// A function block for TcpIp control. Body should be called, 
// but all the logic is done with method calling and awaiting "TRUE" returned when the method finishes.
FUNCTION_BLOCK FB_TcpIpCommControl 
EXTENDS ZigaLibs_Core.FB_HasInstanceNameAndPath 
IMPLEMENTS I_TcpIpCommControl

VAR
	_socketClose			: Tc2_TcpIp.FB_SocketClose;
	_error					: BOOL;
	_errorReceiving			: BOOL;
	_errorSending			: BOOL;
	_isConnected			: BOOL;
	_clientServerControl	: Tc2_TcpIp.FB_ClientServerConnection;
	_socketHandle			: Tc2_TcpIp.T_HSOCKET;
	_logger					: REFERENCE TO ZigaLibs_Logging.I_Logger;
END_VAR

_clientServerControl(nMode := Tc2_TcpIp.CONNECT_MODE_ENABLEDBG, hSocket => _socketHandle);
_error := _errorReceiving OR _errorSending OR _clientServerControl.bError;

// Connets to the target client with the provided Ip address and port
METHOD Connect : BOOL
VAR_INPUT
	Ipv4Address	: Tc2_System.T_IPv4Addr;	// Ip Address
	Port		: UINT;	// Port
END_VAR
VAR_INST
	connected	: R_TRIG;
END_VAR
VAR
	sb	: ZigaLibs_Core.FB_StringBuilder;
END_VAR
connected(CLK := _clientServerControl.eState = Tc2_TcpIp.E_SocketConnectionState.eSOCKET_CONNECTED AND NOT _clientServerControl.bError);
IF connected.Q THEN
	sb.AddString('Connected to')
		.AddWithQuotationMark(_clientServerControl.sRemoteHost)
		.AddString(' with port ')
		.AddAny(_clientServerControl.nRemotePort);
	THIS^.WriteInfoLog(sb.Create());
END_IF

IF THIS^.IsConnected = FALSE THEN
	_clientServerControl.bEnable := TRUE;
	_clientServerControl.sRemoteHost := Ipv4Address;
	_clientServerControl.nRemotePort := Port;
	_clientServerControl.sSrvNetID := '';
ELSE
	Connect := TRUE;
END_IF
END_METHOD

// Disconnects from the server and closes all active socket connections. Returns TRUE when done.
METHOD Disconnect : BOOL
VAR_INST
	disconnected	: Tc2_Standard.F_TRIG;
END_VAR
VAR
	sb			: ZigaLibs_Core.FB_StringBuilder;
END_VAR
disconnected(CLK := _socketClose.bBusy AND NOT _socketClose.bError);
IF disconnected.Q THEN
	sb.AddString('Disconnected from ')
		.AddWithQuotationMark(_clientServerControl.sRemoteHost)
		.AddString(' with port ')
		.AddAny(_clientServerControl.nRemotePort);
	THIS^.WriteInfoLog(sb.Create());
END_IF

IF _clientServerControl.bEnable THEN
	_clientServerControl.bEnable := FALSE;
END_IF

IF NOT _socketClose.bBusy AND (_socketHandle.handle <> 0) THEN
	_socketClose(bExecute := TRUE, sSrvNetId := '', hSocket := _socketHandle);
END_IF
_socketClose(bExecute := FALSE, sSrvNetId := '', hSocket := _socketHandle);
_errorSending := FALSE;
_errorReceiving := FALSE;

Disconnect := NOT _socketClose.bBusy;
END_METHOD

{attribute 'monitoring' := 'call'}
PROPERTY Error : BOOL
GET
Error := _error;
END_GET
END_PROPERTY

METHOD FB_init : BOOL
VAR_INPUT
	bInitRetains 	: BOOL; // if TRUE, the retain variables are initialized (warm start / cold start)
	bInCopyCode 	: BOOL;  // if TRUE, the instance afterwards gets moved into the copy code (online change)
	logger			: REFERENCE TO ZigaLibs_Logging.I_Logger;
END_VAR
_logger REF= logger;
END_METHOD

METHOD GetLogPrefix : STRING
VAR_INPUT
END_VAR
GetLogPrefix := Tc2_Standard.CONCAT(THIS^.InstancePath, ': ');
END_METHOD

{attribute 'monitoring' := 'call'}
PROPERTY PUBLIC IsConnected : BOOL
GET
IsConnected := _clientServerControl.eState = Tc2_TcpIp.E_SocketConnectionState.eSOCKET_CONNECTED;
END_GET
END_PROPERTY

// Awaits a response from the client and returns TRUE when done. Response string can be found in the refResponse
// Method needs to be called untill TRUE is returned to finish the sending sequence!
METHOD Receive : BOOL
VAR_INPUT
	refResponse	: REFERENCE TO Tc2_System.T_MaxString;	// Response will be written to the string variable here
END_VAR
VAR_INST
	sResponse			: Tc2_System.T_MaxString;
	eSocketReceiveState	: E_SocketReceiveState;
	fbSocketReceive		: Tc2_TcpIp.FB_SocketReceive;
	bReceiveError		: BOOL;
END_VAR
VAR
	sb	: ZigaLibs_Core.FB_StringBuilder;
END_VAR
CASE eSocketReceiveState OF
	E_SocketReceiveState.READY:
		fbSocketReceive(bExecute := FALSE);
		IF THIS^.IsConnected THEN
			bReceiveError := FALSE;
			fbSocketReceive(
				bExecute := TRUE,
				cbLen := SIZEOF(refResponse),
				pDest := ADR(refResponse),
				sSrvNetId := '',
				hSocket := _socketHandle);
			eSocketReceiveState := E_SocketReceiveState.RECEIVING;
		END_IF
	
	E_SocketReceiveState.RECEIVING:
		fbSocketReceive(bExecute := FALSE);
		IF NOT fbSocketReceive.bError AND_THEN NOT fbSocketReceive.bBusy THEN
			eSocketReceiveState := E_SocketReceiveState.DONE;
		ELSIF fbSocketReceive.bError THEN
			eSocketReceiveState := E_SocketReceiveState.ERROR;	
		END_IF
	
	E_SocketReceiveState.DONE:
		Receive := TRUE;
		eSocketReceiveState := E_SocketReceiveState.READY;
	
	E_SocketReceiveState.ERROR:
		bReceiveError := TRUE;
		eSocketReceiveState := E_SocketReceiveState.DONE;
		
		sb.AddString('Error while receiving from ')
			.AddWithDblQuotationMarks(_socketHandle.remoteAddr.sAddr)
			.AddString('. Error code received is ')
			.AddWithQuotationMark(TO_STRING(fbSocketReceive.nErrId));
		THIS^.WriteErrorLog(sb.Create());
END_CASE

_errorReceiving := bReceiveError;
END_METHOD

{attribute 'monitoring' := 'call'}
(* Gets or sets the reconnect period. 
The value should not be set too low, since timeout periods of > 30 s may occur in the event of a network interruption. 
If the value is too low, command execution would be interrupted prematurely, and ADS error code 1861 (timeout elapsed) 
would be returned instead of the Winsocket error WSAETIMEDOUT.*)
PROPERTY PUBLIC ReconnectPeriod : TIME
GET
ReconnectPeriod := _clientServerControl.tReconnect;
END_GET
SET
IF ReconnectPeriod > T#30S THEN
	_clientServerControl.tReconnect := ReconnectPeriod;
END_IF
END_SET
END_PROPERTY

// Sends the command to the client and returns TRUE when done. 
// Method needs to be called untill TRUE is returned to finish the sending sequence!
METHOD Send : BOOL
VAR_INPUT
	sCommand	: Tc2_System.T_MaxString;	// Command to be send
END_VAR
VAR_INST
	fbSocketSend		: Tc2_TcpIp.FB_SocketSend;
	eSsocketSendState	: E_SocketSendState;
	arrSendDataBytes	: ARRAY[0..255] OF BYTE;
	nSendDataCount		: UDINT;
	bSendError			: BOOL;
END_VAR

VAR
	sb	: ZigaLibs_Core.FB_StringBuilder;
END_VAR
CASE eSsocketSendState OF
	E_SocketSendState.READY:
		bSendError := FALSE;
		IF sCommand <> '' THEN
			// Clear array for new data
			Tc2_System.MEMSET(
				destAddr := ADR(arrSendDataBytes),
				n := SIZEOF(arrSendDataBytes),
				fillByte := 0);
				
			// Prepare data
			Tc2_System.MEMCPY(
				destAddr := ADR(arrSendDataBytes),
				n := SIZEOF(sCommand),
				srcAddr := ADR(sCommand));
				
			// Get the data count, no empty bytes
			nSendDataCount := 0;
			FOR nSendDataCount := 0 TO SIZEOF(arrSendDataBytes) BY 1 DO
				IF arrSendDataBytes[nSendDataCount] = 0 THEN
					EXIT;
				END_IF
			END_FOR

			// Send data
			fbSocketSend(
				bExecute := TRUE,
				cbLen := nSendDataCount,
				pSrc := ADR(arrSendDataBytes),
				hSocket := _socketHandle);
				
			eSsocketSendState := E_SocketSendState.SENDING;
		END_IF
	
	E_SocketSendState.SENDING:
		fbSocketSend(bExecute := FALSE);
		IF fbSocketSend.bError THEN 
			eSsocketSendState := E_SocketSendState.ERROR;
		ELSIF fbSocketSend.bBusy = FALSE THEN
				eSsocketSendState := E_SocketSendState.DONE;
		END_IF
		
	E_SocketSendState.DONE:
		Send := TRUE;
		eSsocketSendState := E_SocketSendState.READY;
		
	E_SocketSendState.ERROR:
		bSendError := TRUE;
		eSsocketSendState := E_SocketSendState.DONE;
		sb.AddString('Error while sending from ')
			.AddWithQuotationMark(_socketHandle.localAddr.sAddr)
			.AddString(' to ')
			.AddWithDblQuotationMarks(_socketHandle.remoteAddr.sAddr)
			.AddString('. Command being sent was ')
			.AddWithQuotationMark(sCommand)
			.AddString('. Error code received is ')
			.AddWithQuotationMark(TO_STRING(fbSocketSend.nErrId));
		THIS^.WriteErrorLog(sb.Create());
		
END_CASE

_errorSending := bSendError;
END_METHOD

METHOD WriteErrorLog
VAR_INPUT
	message	: Tc2_System.T_MaxString;
END_VAR
IF NOT __ISVALIDREF(_logger) THEN
	RETURN;
END_IF

_logger.LogError(Tc2_Standard.CONCAT(THIS^.GetLogPrefix(), (message)));
END_METHOD

METHOD WriteInfoLog
VAR_INPUT
	message	: Tc2_System.T_MaxString;
END_VAR
IF NOT __ISVALIDREF(_logger) THEN
	RETURN;
END_IF

_logger.LogInfo(Tc2_Standard.CONCAT(THIS^.GetLogPrefix(), (message)));
END_METHOD

END_FUNCTION_BLOCK

(* stored: Version 1.1.0.1, ProductVersion 3.1.4024.15
   POU FB_TcpIpCommControl: Id {c1a18772-55c5-40c9-9a81-d2bef65ca48e}, SpecialFunc None
   Folder Constructor: Id {8e03ba55-7e0e-08dc-121d-63148ed4730e}
   Folder Private: Id {2efa374f-f01f-026b-1d46-811c1330f5ed}
   Folder Methods: Id {e8932037-c29c-0039-0710-e32b2dab25e8}
   Folder Public: Id {fad2bedc-c621-0e7a-10b3-e31e1f06606d}
   Folder Methods: Id {ca322448-3c94-05d4-3845-31017722f3e8}
   Folder Properties: Id {22abed52-9456-006d-1b18-e9ce2512ef08}
   Method Connect: Id {dd6866c4-171a-4bfc-95da-36f23ef555cb}
   Method Disconnect: Id {ed43bf91-0d1a-4937-b486-9810fb451075}
   Property Error: Id {5c00ee02-56f4-43bb-9e23-9bd70a569756}
   Get Get: Id {6ff5fc3c-9cf5-40c2-8121-3ea148df9e2e}
   Method FB_init: Id {7ffdea42-4472-0096-2bdd-6e582451a91a}
   Method GetLogPrefix: Id {18ab9aea-3da0-09f1-3eba-322fd828d465}
   Property IsConnected: Id {5e9ad8a1-6ad5-4c8b-a48a-e8e88fb474a1}
   Get Get: Id {d7cb8efd-ba1c-4704-9fa9-84315798b314}
   Method Receive: Id {7a2e245a-21db-4c97-a338-d1db7e183060}
   Property ReconnectPeriod: Id {960f0c0e-a8f0-4b6e-8253-4e69f0060513}
   Get Get: Id {873b00e4-9119-45cc-8128-e1136d45c726}
   Set Set: Id {6a4a98a9-2fc1-42f2-81eb-5c784556b477}
   Method Send: Id {e24d3e99-79a0-4664-a580-6ca5668718f9}
   Method WriteErrorLog: Id {73b3d1d9-35e8-0cdd-1254-94fd3c0ce0ac}
   Method WriteInfoLog: Id {5261de02-aff5-0ae2-3636-4265a63b170c} *)
